Yaskawa INFORM job: FRONT_WELD_180ST_5040_1.JBI

/JOB
//NAME FRONT_WELD_180ST_5040_1
///FOLDERNAME 02-SKRZYNIE_JOBS
//POS
///NPOS 32,32,0,2,0,0
///TOOL 0
///POSTYPE PULSE
///PULSE
C00000=0,-52280,40443,0,6876,0
C00001=252,-53930,13084,-98,24463,-31882
C00002=-30875,-45817,-9234,13562,36212,-43234
C00003=-78118,-33412,-6590,31148,62743,-59116
C00004=-95672,-18401,-524,43648,77081,-65694
C00005=-95672,-18401,-524,43648,77081,-65694
C00006=-57798,-21642,-871,33514,39109,-45911
C00007=-51167,-14064,3513,23793,42928,-41031
C00008=-41740,-17885,366,19270,39899,-37217
C00009=-34149,-20360,-1601,15004,37885,-33849
C00010=-27563,-22213,-3010,10883,36465,-30729
C00011=-42487,-35877,-10644,41507,25485,-46082
C00012=-95672,-18401,-524,43648,77081,-65694
C00013=-95672,-18401,-524,43648,77081,-65694
C00014=-79329,-40248,-13867,46310,64370,-64671
C00015=0,-40093,13463,3,15613,-32000
C00016=0,-39212,13596,-3,16186,32000
C00017=36805,-50815,-6409,-18927,30678,47791
C00018=95672,-18401,-524,-43648,77081,65694
C00019=95672,-18401,-524,-43648,77081,65694
C00020=57798,-21642,-871,-33514,39109,45911
C00021=50153,-15754,4668,-25993,39511,41697
C00022=41002,-19349,1638,-21216,36461,37821
C00023=31100,-21858,-285,-14912,33842,33092
C00024=25317,-23265,-1354,-10729,32660,30092
C00025=42487,-35877,-10644,-41507,25485,46082
C00026=95672,-18401,-524,-43648,77081,65694
C00027=101139,-20014,-1807,-43255,79399,67016
C00028=81889,-36590,-12546,-37164,67407,61636
C00029=0,-45421,13373,-5,11660,32001
C00030=-252,-53930,13084,98,24463,31882
C00031=0,-52280,40443,0,6876,0
BC00000=801491
BC00001=813034
BC00002=879617
BC00003=896376
BC00004=908397
BC00005=941160
BC00006=935162
BC00007=935162
BC00008=935162
BC00009=935162
BC00010=935162
BC00011=935162
BC00012=941160
BC00013=908397
BC00014=908397
BC00015=870737
BC00016=870737
BC00017=878086
BC00018=908397
BC00019=941160
BC00020=935162
BC00021=935162
BC00022=935162
BC00023=935162
BC00024=935162
BC00025=935162
BC00026=941160
BC00027=908397
BC00028=902485
BC00029=870737
BC00030=813034
BC00031=801491
///POSTYPE BASE
///RECTAN
///RCONF 0,0,0,0,0,0,0,0,0,0,0,0,0,0,0,0,0,0,0,0,0,0,0,0
P00400=5.920,-3.503,-0.024,0.0000,0.0000,0.0000
P00401=3.430,-0.021,1.131,0.0000,0.0000,0.0000
//INST
///DATE 2024/05/14 12:59
///ATTR SC,RW
///GROUP1 RB1,BS1
NOP
MOVJ C00000 BC00000 VJ=20.00
MOVJ C00001 BC00001 VJ=20.00
MOVJ C00002 BC00002 VJ=15.00
MOVJ C00003 BC00003 VJ=15.00
MOVJ C00004 BC00004 VJ=15.00
MOVJ C00005 BC00005 VJ=20.00
'------------------------
'W32
'------------------------
MOVL C00006 BC00006 V=500.0
SFTON P0400
MOVL C00007 BC00007 V=66.7 PL=0
MACRO1 MJ#(0) ARGF14
ARCON
MOVL C00008 BC00008 V=10.0
MOVL C00009 BC00009 V=10.0
MOVL C00010 BC00010 V=10.0
ARCOF
SFTOF
MOVL C00011 BC00011 V=166.7
MOVJ C00012 BC00012 VJ=20.00
MOVJ C00013 BC00013 VJ=20.00
MOVJ C00014 BC00014 VJ=20.00
MOVJ C00015 BC00015 VJ=15.00
MOVJ C00016 BC00016 VJ=10.00
MOVJ C00017 BC00017 VJ=15.00
MOVJ C00018 BC00018 VJ=10.00
MOVJ C00019 BC00019 VJ=15.00
'------------------------
'W33
'------------------------
MOVL C00020 BC00020 V=500.0
SFTON P0401
MOVL C00021 BC00021 V=66.7 PL=0
MACRO1 MJ#(0) ARGF14
ARCON
MOVL C00022 BC00022 V=10.0
MOVL C00023 BC00023 V=10.0
MOVL C00024 BC00024 V=10.0
ARCOF
SFTOF
MOVL C00025 BC00025 V=166.7
MOVJ C00026 BC00026 VJ=10.00
MOVJ C00027 BC00027 VJ=10.00
MOVJ C00028 BC00028 VJ=10.00
MOVJ C00029 BC00029 VJ=15.00
MOVJ C00030 BC00030 VJ=30.00
MOVJ C00031 BC00031 VJ=40.00
END
